TYPE ASCF_CC_OPCUACS_Writer_Temp_String :
STRUCT
	stReadListReturnInfo	: ARRAY [1..1] OF ST_UAReadListReturnInfo;
	Value		: STRING		:= '';
END_STRUCT
END_TYPE

(* stored: Version 1.1.0.1, ProductVersion 3.1.4026.4
   DUT ASCF_CC_OPCUACS_Writer_Temp_String: Id {9849ebdd-0ec7-4dba-a9f0-3b1113887209} *)
